{attribute addProperty BoxType "EL3773-0000-0016"}
{attribute addProperty Id "U2_SAMPLESAT %I*ARRAY [1..10] OF INT16020"}
{attribute addProperty CRC "3265976639"}
{attribute addProperty SizeInBites "160"}
{attribute addProperty SizeInBytes "20"}
TYPE L2_Voltage_Samples_C2AAD93F :
STRUCT
	{attribute addProperty Name "U2_SAMPLES"}
	U2_SAMPLES AT %I* : ARRAY [1..10] OF INT;
END_STRUCT
END_TYPE

(* stored: Version 1.2.0.0, ProductVersion 3.1.4024.9
   DUT L2_Voltage_Samples_C2AAD93F: Id {66a3206e-b00e-4eb4-80d0-8fe4906f8cce} *)
